FUNCTION_BLOCK ATURNTABLE_MUX (* Composite FB wrapping other FBs *)
  (* Standard: 61499-2 *)
  (* Version 0.0, 2008-07-10, 4DIAC-IDE, 4DIAC-Consortium *)
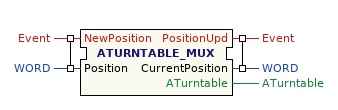
  EVENT_INPUT
    NewPosition WITH Position; (* Confirmation from Plug *)
  END_EVENT
  EVENT_OUTPUT
    PositionUpd WITH CurrentPosition; (* Request from Socket *)
  END_EVENT
  VAR_INPUT
    Position : WORD; (* Confirmation Data from Plug *)
  END_VAR
  VAR_OUTPUT
    CurrentPosition : WORD; (* Request Data from Socket *)
  END_VAR
  PLUGS
    ATurntable : ATurntable;
  END_PLUGS
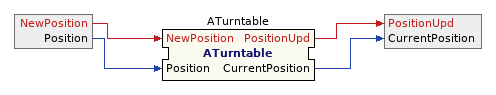
  EVENT_CONNECTIONS
    NewPosition TO ATurntable.NewPosition;
    ATurntable.PositionUpd TO PositionUpd;
  END_CONNECTIONS
  DATA_CONNECTIONS
    Position TO ATurntable.Position;
    ATurntable.CurrentPosition TO CurrentPosition;
  END_CONNECTIONS
END_FUNCTION_BLOCK
